TYPE (* logiBUS DI Struct Octal *)
  (* Version 1.0, 2026-05-28, franz *)
  PACKAGE logiBUS::io::DI;
  IMPORT eclipse4diac::core::TypeHash;
  IMPORT logiBUS::io::DI::logiBUS_DI_S;
  logiBUS_DI_S_Octal : STRUCT
    Port1 : logiBUS_DI_S := (Pin := 255);
    Port2 : logiBUS_DI_S := (Pin := 255);
    Port3 : logiBUS_DI_S := (Pin := 255);
    Port4 : logiBUS_DI_S := (Pin := 255);
    Port5 : logiBUS_DI_S := (Pin := 255);
    Port6 : logiBUS_DI_S := (Pin := 255);
    Port7 : logiBUS_DI_S := (Pin := 255);
    Port8 : logiBUS_DI_S := (Pin := 255);
  END_STRUCT;
END_TYPE
